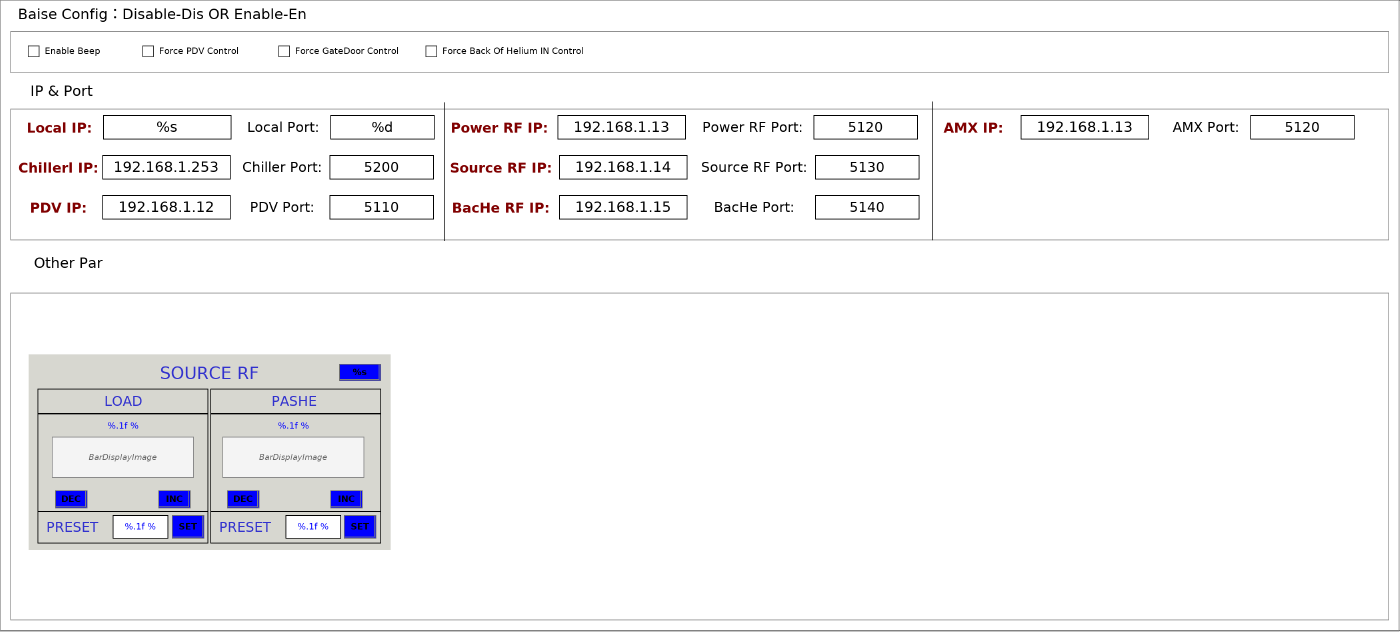
VISUALIZATION Config_Base  // 1750x790
    Group (0,0 1751x0)
        Line (0,788) (1750,788)
        Line (0,0) (0,782)
        Line (0,0) (1750,0)
        Line (1750,0) (1750,782)
    GroupBox (13,358 1723x417)
        Label (-2382,-64 501x61), "参数设置说明"
        Label (-2397,-19 522x195), "需切换界面左上角控制模式为“配置模式”，根据参数栏 左上方提示内容及其设置框说明标题，设置相应的参数并按 “保存配置”按钮3秒以上，直到右侧黄灯闪烁 设置完成参数后需根据相应需求选择对应控制模式"
        RoundedRectangle (23,85 452x244), colour toggle: NOT FuncModule_RS232_SRF.serialConnected
        Rectangle (250,159 213x162)
        Rectangle (34,159 213x162)
        Label (153,93 192x31), "SOURCE RF"
        RoundedRectangle (34,281 213x40)
        Label (42,290 85x22), "PRESET"
        RoundedRectangle (128,286 69x29), "%.1f %", text variable: FuncModule_RS232_SRF.goPosLoad, input disabled if: TRUE
            OnMouseClick: write the text variable via Default, min 0.0, max 100.0
        Button (56,255 40x22), "DEC", input disabled if: TRUE
            OnMouseClick: execute { FuncModule_RS232_SRF.LoadDEC(); }
        Button (185,255 40x22), "INC", input disabled if: TRUE
            OnMouseClick: execute { FuncModule_RS232_SRF.LoadINC(); }
        Button (271,255 40x22), "DEC", input disabled if: TRUE
            OnMouseClick: execute { FuncModule_RS232_SRF.PhaseDEC(); }
        Button (400,255 40x22), "INC", input disabled if: TRUE
            OnMouseClick: execute { FuncModule_RS232_SRF.PhaseINC(); }
        Button (202,286 40x29), "SET", input disabled if: TRUE
            OnMouseClick: execute { FuncModule_RS232_SRF.LoadAndPhaseGo(); }
        RoundedRectangle (250,281 213x40)
        Label (258,290 85x22), "PRESET"
        RoundedRectangle (344,286 69x29), "%.1f %", text variable: FuncModule_RS232_SRF.goPosPhase, input disabled if: TRUE
            OnMouseClick: write the text variable via Default, min 0.0, max 100.0
        Button (417,286 40x29), "SET", input disabled if: TRUE
            OnMouseClick: execute { FuncModule_RS232_SRF.LoadAndPhaseGo(); }
        Rectangle (34,128 213x31)
        Label (109,133 65x21), "LOAD"
        Rectangle (250,128 213x31)
        Label (315,133 80x21), "PASHE"
        Button (411,97 52x21), "%s", text variable: FuncModule_RS232_SRF.rec_MAStr, input disabled if: TRUE
            OnMouseClick: execute { FuncModule_RS232_SRF.ManulORAuto(); }
        BarDisplayImage (52,188 177x51), value: FuncModule_RS232_SRF.load, style: BarDisplayImage-Gray, scale format: %.1f, scale 0..100
        BarDisplayImage (265,188 177x51), value: FuncModule_RS232_SRF.phase, style: BarDisplayImage-Gray, scale format: %.1f, scale 0..100
        RoundedRectangle (113,160 56x29), "%.1f %", text variable: FuncModule_RS232_SRF.load, colour toggle: FuncModule_RS232_SRF.loadRunErr
        RoundedRectangle (326,160 56x29), "%.1f %", text variable: FuncModule_RS232_SRF.phase, colour toggle: FuncModule_RS232_SRF.phashRunErr
    Label (1928,1052 45x20)
    Label (5,3 396x30), "Baise Config：Disable-Dis OR Enable-En"
    Label (5,99 144x30), "IP & Port"
    GroupBox (13,31 1723x60)
        Label (-2382,-64 501x61), "参数设置说明"
        Label (-2397,-19 522x195), "需切换界面左上角控制模式为“配置模式”，根据参数栏 左上方提示内容及其设置框说明标题，设置相应的参数并按 “保存配置”按钮3秒以上，直到右侧黄灯闪烁 设置完成参数后需根据相应需求选择对应控制模式"
        Checkbox (20,13 116x40), "Enable Beep", variable: fbMachineState.HMI_EnableBuzzer
        Checkbox (163,13 152x40), "Force PDV Control", variable: gEnablePDVOpenClose
        Checkbox (333,13 175x40), "Force GateDoor Control", variable: gEnableGDOpenClose
        Checkbox (517,13 224x40), "Force Back Of Helium IN Control", variable: gEnableHeInOpenClose
    GroupBox (13,128 1723x172)
        Label (-2382,-64 501x61), "参数设置说明"
        Label (-2397,-19 522x195), "需切换界面左上角控制模式为“配置模式”，根据参数栏 左上方提示内容及其设置框说明标题，设置相应的参数并按 “保存配置”按钮3秒以上，直到右侧黄灯闪烁 设置完成参数后需根据相应需求选择对应控制模式"
        Label (9,16 105x32), "Local IP:"
        Rectangle (116,16 160x30), "%s", text variable: gLocalHostIp, input disabled if: NOT (gRunningState=RunningStatus.eManualState AND gCtrlMode=ControlMode.eConfig)
        Rectangle (400,16 130x30), "%d", text variable: gLocalHostPort, input disabled if: NOT (gRunningState=RunningStatus.eManualState AND gCtrlMode=ControlMode.eConfig)
        Label (287,16 108x30), "Local Port:"
        Label (8,66 105x32), "Chillerl IP:"
        Label (8,116 105x32), "PDV IP:"
        Label (541,16 141x32), "Power RF IP:"
        Label (543,66 141x32), "Source RF IP:"
        Label (543,116 141x32), "BacHe RF IP:"
        Rectangle (1550,16 130x30), "5120", text variable: gLocalHostPort, input disabled if: NOT (gRunningState=RunningStatus.eManualState AND gCtrlMode=ControlMode.eConfig)
    Label (20,311 131x36), "Other Par"
    Rectangle (128,194 160x30), "192.168.1.253", text variable: gLocalHostIp, input disabled if: NOT (gRunningState=RunningStatus.eManualState AND gCtrlMode=ControlMode.eConfig)
    Rectangle (412,194 130x30), "5200", text variable: gLocalHostPort, input disabled if: NOT (gRunningState=RunningStatus.eManualState AND gCtrlMode=ControlMode.eConfig)
    Label (299,194 108x30), "Chiller Port:"
    Rectangle (128,244 160x30), "192.168.1.12", text variable: gLocalHostIp, input disabled if: NOT (gRunningState=RunningStatus.eManualState AND gCtrlMode=ControlMode.eConfig)
    Rectangle (412,244 130x30), "5110", text variable: gLocalHostPort, input disabled if: NOT (gRunningState=RunningStatus.eManualState AND gCtrlMode=ControlMode.eConfig)
    Label (299,244 108x30), "PDV Port:"
    Rectangle (697,144 160x30), "192.168.1.13", text variable: gLocalHostIp, input disabled if: NOT (gRunningState=RunningStatus.eManualState AND gCtrlMode=ControlMode.eConfig)
    Rectangle (1017,144 130x30), "5120", text variable: gLocalHostPort, input disabled if: NOT (gRunningState=RunningStatus.eManualState AND gCtrlMode=ControlMode.eConfig)
    Label (868,144 146x30), "Power RF Port:"
    Rectangle (699,194 160x30), "192.168.1.14", text variable: gLocalHostIp, input disabled if: NOT (gRunningState=RunningStatus.eManualState AND gCtrlMode=ControlMode.eConfig)
    Rectangle (1019,194 130x30), "5130", text variable: gLocalHostPort, input disabled if: NOT (gRunningState=RunningStatus.eManualState AND gCtrlMode=ControlMode.eConfig)
    Label (870,194 146x30), "Source RF Port:"
    Rectangle (699,244 160x30), "192.168.1.15", text variable: gLocalHostIp, input disabled if: NOT (gRunningState=RunningStatus.eManualState AND gCtrlMode=ControlMode.eConfig)
    Rectangle (1019,244 130x30), "5140", text variable: gLocalHostPort, input disabled if: NOT (gRunningState=RunningStatus.eManualState AND gCtrlMode=ControlMode.eConfig)
    Label (870,244 146x30), "BacHe Port:"
    Label (1160,144 114x32), "AMX IP:"
    Rectangle (1276,144 160x30), "192.168.1.13", text variable: gLocalHostIp, input disabled if: NOT (gRunningState=RunningStatus.eManualState AND gCtrlMode=ControlMode.eConfig)
    Label (1455,144 105x30), "AMX Port:"
    Line (556,301) (556,128)
    Line (1166,300) (1166,127)
END_VISUALIZATION

(* stored: Version 1.1.0.1, ProductVersion 3.1.4024.12
   Visu Config_Base: Id {f9ce4674-9bb4-44a4-92c7-d50e4d417430} *)
